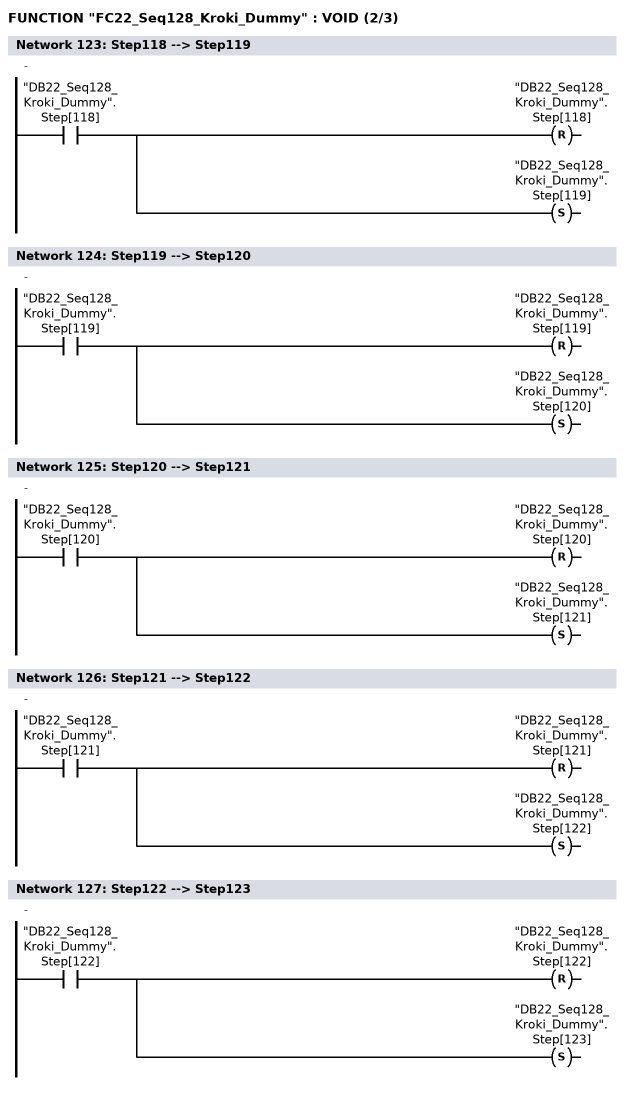
      A     "DB22_Seq128_Kroki_Dummy".Step[118];
      R     "DB22_Seq128_Kroki_Dummy".Step[118];
      S     "DB22_Seq128_Kroki_Dummy".Step[119];

NETWORK
TITLE = Step119 --> Step120
//-
      A     "DB22_Seq128_Kroki_Dummy".Step[119];
      R     "DB22_Seq128_Kroki_Dummy".Step[119];
      S     "DB22_Seq128_Kroki_Dummy".Step[120];

NETWORK
TITLE = Step120 --> Step121
//-
      A     "DB22_Seq128_Kroki_Dummy".Step[120];
      R     "DB22_Seq128_Kroki_Dummy".Step[120];
      S     "DB22_Seq128_Kroki_Dummy".Step[121];

NETWORK
TITLE = Step121 --> Step122
//-
      A     "DB22_Seq128_Kroki_Dummy".Step[121];
      R     "DB22_Seq128_Kroki_Dummy".Step[121];
      S     "DB22_Seq128_Kroki_Dummy".Step[122];

NETWORK
TITLE = Step122 --> Step123
//-
      A     "DB22_Seq128_Kroki_Dummy".Step[122];
      R     "DB22_Seq128_Kroki_Dummy".Step[122];
      S     "DB22_Seq128_Kroki_Dummy".Step[123];

NETWORK
TITLE = Step123 --> Step124
//-
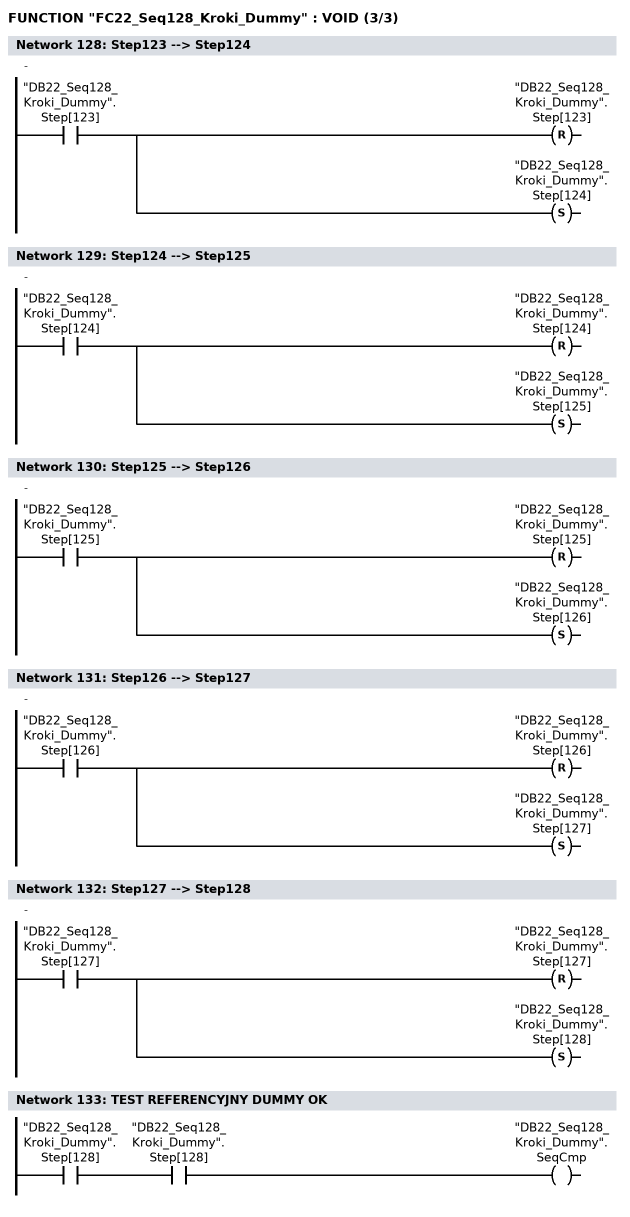
      A     "DB22_Seq128_Kroki_Dummy".Step[123];
      R     "DB22_Seq128_Kroki_Dummy".Step[123];
      S     "DB22_Seq128_Kroki_Dummy".Step[124];
NETWORK
TITLE = Step124 --> Step125
//-
      A     "DB22_Seq128_Kroki_Dummy".Step[124];
      R     "DB22_Seq128_Kroki_Dummy".Step[124];
      S     "DB22_Seq128_Kroki_Dummy".Step[125];

NETWORK
TITLE = Step125 --> Step126
//-
      A     "DB22_Seq128_Kroki_Dummy".Step[125];
      R     "DB22_Seq128_Kroki_Dummy".Step[125];
      S     "DB22_Seq128_Kroki_Dummy".Step[126];

NETWORK
TITLE = Step126 --> Step127
//-
      A     "DB22_Seq128_Kroki_Dummy".Step[126];
      R     "DB22_Seq128_Kroki_Dummy".Step[126];
      S     "DB22_Seq128_Kroki_Dummy".Step[127];

NETWORK
TITLE = Step127 --> Step128
//-
      A     "DB22_Seq128_Kroki_Dummy".Step[127];
      R     "DB22_Seq128_Kroki_Dummy".Step[127];
      S     "DB22_Seq128_Kroki_Dummy".Step[128];

NETWORK
TITLE =TEST REFERENCYJNY DUMMY OK

      A     "DB22_Seq128_Kroki_Dummy".Step[128];

      A     "DB22_Seq128_Kroki_Dummy".Step[128];
      =     "DB22_Seq128_Kroki_Dummy".SeqCmp;

END_FUNCTION

